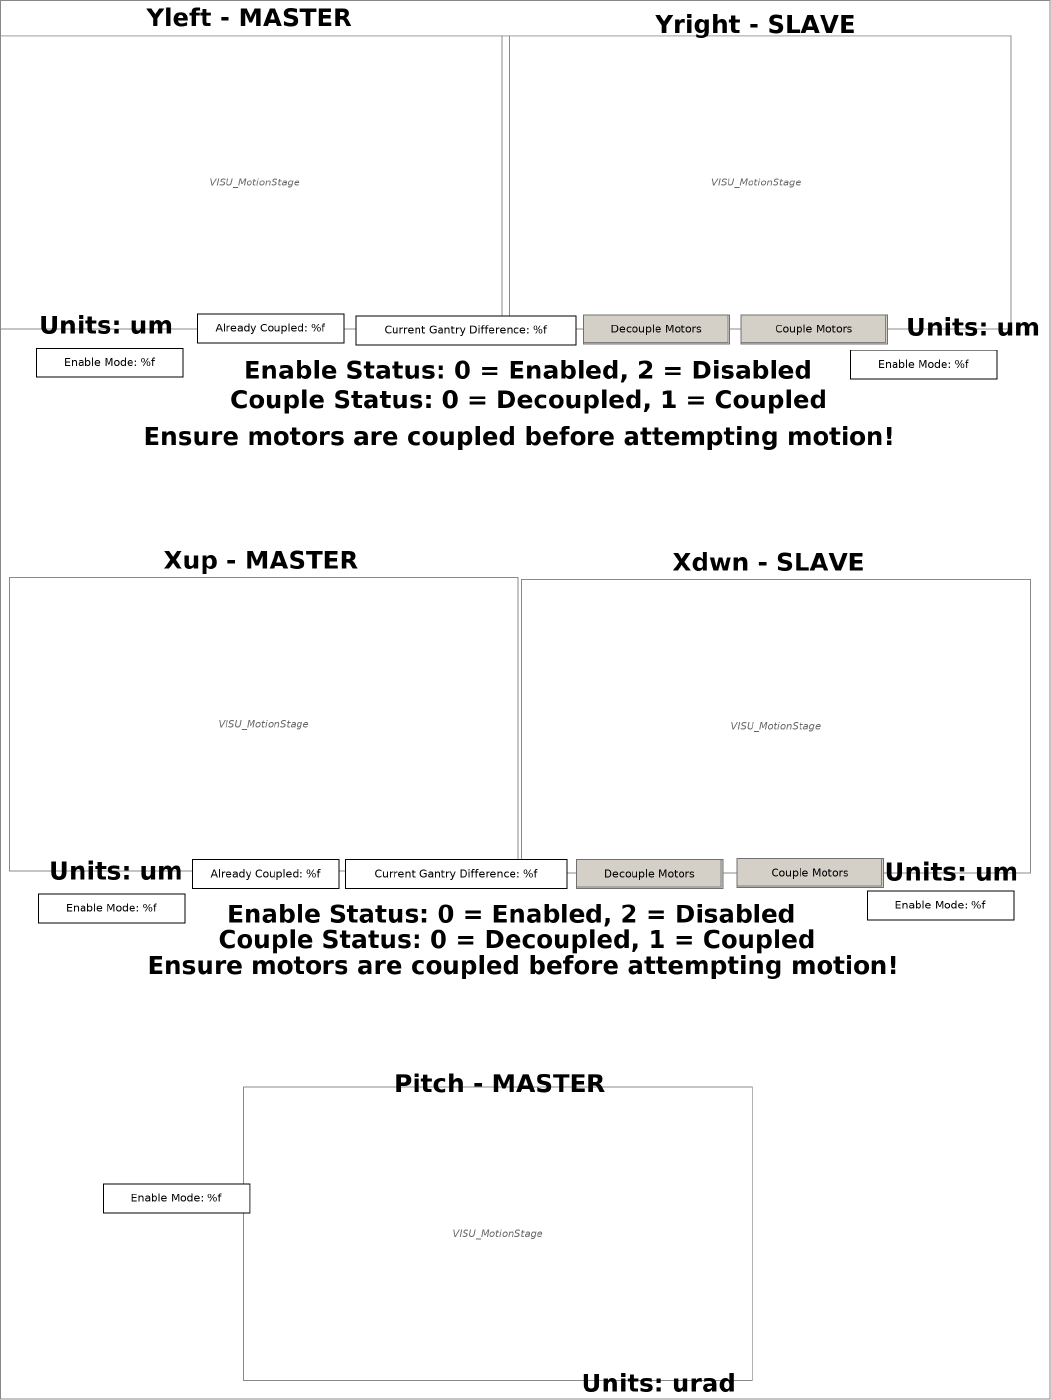
VISUALIZATION Visualization  // 1073x1429
    Label (14,2 481x31), "Yleft - MASTER"
    Frame (0,36 520x300)
        shows VISU_MotionStage(VisuMotionStage := GVL_M2L0.M7, Extras := GVL_M2L0.M7_Extras)
    Frame (512,36 520x300)
        shows VISU_MotionStage(VisuMotionStage := GVL_M2L0.M8, Extras := GVL_M2L0.M8_Extras)
    Label (531,9 481x31), "Yright - SLAVE"
    Rectangle (201,320 150x30), "Already Coupled: %f", tooltip "Couple Status: TRUE if coupled", text variable: Main.M2L0.bGantryAlreadyCoupledY
    Rectangle (363,322 225x30), "Current Gantry Difference: %f", tooltip "Current Gantry Difference in um", text variable: Main.M2L0.fCurrGantryY_um
    Button (756,321 150x30), "Couple Motors", tooltip "Press To Couple Motors"
        OnMouseDown: execute { Main.M2L0.bExecuteCoupleY := TRUE; }
    Frame (9,589 520x300)
        shows VISU_MotionStage(VisuMotionStage := GVL_M2L0.M9, Extras := GVL_M2L0.M9_Extras)
    Label (26,556 481x31), "Xup - MASTER"
    Frame (532,591 520x300)
        shows VISU_MotionStage(VisuMotionStage := GVL_M2L0.M10, Extras := GVL_M2L0.M10_Extras)
    Label (544,558 481x31), "Xdwn - SLAVE"
    Rectangle (196,877 150x30), "Already Coupled: %f", tooltip "Couple Status: TRUE if coupled", text variable: Main.M2L0.bGantryAlreadyCoupledX
    Rectangle (352,877 227x30), "Current Gantry Difference: %f", tooltip "Current Gantry Difference in um", text variable: Main.M2L0.fCurrGantryX_um
    Frame (248,1109 520x300)
        shows VISU_MotionStage(VisuMotionStage := GVL_M2L0.M11, Extras := GVL_M2L0.M11_Extras)
    Label (270,1090 481x31), "Pitch - MASTER"
    Label (31,316 155x31), "Units: um"
    Label (916,318 155x31), "Units: um"
    Label (41,873 155x31), "Units: um"
    Label (894,874 155x31), "Units: um"
    Label (595,1396 155x31), "Units: urad"
    Rectangle (37,355 150x30), "Enable Mode: %f", tooltip "Write 0 to Enable, 2 to Disable", text variable: GVL_M2L0.M7.nEnableMode
    Rectangle (868,357 150x30), "Enable Mode: %f", tooltip "Write 0 to Enable, 2 to Disable", text variable: GVL_M2L0.M8.nEnableMode
    Button (595,321 150x30), "Decouple Motors", tooltip "Press To Decouple Motors for independent control"
        OnMouseDown: execute { Main.M2L0.bExecuteDecoupleY := TRUE; }
    Button (588,877 150x30), "Decouple Motors", tooltip "Press To Decouple Motors for independent control"
        OnMouseDown: execute { Main.M2L0.bExecuteDecoupleX := TRUE; }
    Button (752,876 150x30), "Couple Motors", tooltip "Press To Couple Motors"
        OnMouseDown: execute { Main.M2L0.bExecuteCoupleX := TRUE; }
    Rectangle (39,912 150x30), "Enable Mode: %f", tooltip "Write 0 to Enable, 2 to Disable", text variable: GVL_M2L0.M9.nEnableMode
    Rectangle (885,909 150x30), "Enable Mode: %f", tooltip "Write 0 to Enable, 2 to Disable", text variable: GVL_M2L0.M10.nEnableMode
    Rectangle (105,1208 150x30), "Enable Mode: %f", tooltip "Write 0 to Enable, 2 to Disable", text variable: GVL_M2L0.M11.nEnableMode
    Label (255,362 568x31), "Enable Status: 0 = Enabled, 2 = Disabled"
    Label (247,392 586x31), "Couple Status: 0 = Decoupled, 1 = Coupled"
    Label (238,917 568x31), "Enable Status: 0 = Enabled, 2 = Disabled"
    Label (235,943 586x31), "Couple Status: 0 = Decoupled, 1 = Coupled"
    Label (150,430 760x30), "Ensure motors are coupled before attempting motion!"
    Label (154,970 760x30), "Ensure motors are coupled before attempting motion!"
END_VISUALIZATION

(* stored: Version 1.1.0.1, ProductVersion 3.1.4022.18
   Visu Visualization: Id {af2f16f4-e7e7-4019-a84a-cc323e4115d2} *)
